(*
TIME		: 2023-11-13 14:59
Version		: 1.0
Creator		: Ulysses
Reference	: IOTA - BLUE
Commecnts	: 按钮功能块，总体和Input差不多，针对按钮做了功能的完善。可以将输入信号强制、反转或延迟
*)
(* 不带延迟 *)
Q			:= ((RawIn OR Force) XOR Invert) AND Enable;
rTrig(CLK:= Q);
Q_RT		:= rTrig.Q;
fTrig(CLK:= Q);
Q_FT		:= fTrig.Q;
Q_Tog	:= NOT (TrigOff AND Enable) AND (Q_RT XOR Q_Tog OR (TrigOn AND Enable));
(* 带延迟 *)
tonDelay(IN:= Q, PT:= DelayTime);
Q_Delay		:= tonDelay.Q;
rTrig_Delay(CLK:= Q_Delay);
Q_Delay_RT	:= rTrig_Delay.Q;
fTrig_Delay(CLK:= Q_Delay);
Q_Delay_FT	:= fTrig_Delay.Q;

Q_Delay_Tog := NOT (TrigOffDelay AND Enable) AND (Q_Delay_RT XOR Q_Delay_Tog OR (TrigOnDelay AND Enable));

END_FUNCTION_BLOCK

// ---- TF11PlcSystem/IO/DI_Input.TcPOU
{attribute 'no_check'}
(* 
按钮功能块 Button
按钮功能块，总体和Input差不多，针对按钮做了功能的完善可以将输入信号强制、反转或延迟
*)
FUNCTION_BLOCK DI_Input
VAR_INPUT
	Invert : BOOL := FALSE; (* False: 不反转Direct \ True: 在源头反转输入Invert Input *)
	ForceOn : BOOL; (* 将输入强制为True, Force the In signal to True *)
	ForceOff : BOOL; (* 将输入强制为True, Force the In signal to True *)
	DelayTime : TIME := T#50MS; (* 延迟输出时间，T#0MS代表无延迟，也可充当滤波功能 *)
	LED AT%Q* : BOOL; (* 如果按钮有LED，绑定到LED的输出上，功能块内部本身不控制LED，需要外部程序通过该输入引脚控制 *)
END_VAR
VAR_OUTPUT
	Q : BOOL;(* 直接输出信号 *)
	QRT : BOOL;(* 输入信号的上升沿 *)
	QFT : BOOL;(* 输入信号的下降沿 *)
	RawIn AT%I* :BOOL; (* 原始输入信号，未经强制、反转及延时 *) 
END_VAR
VAR
	rTrig, rTrig_Delay : R_TRIG;
	fTrig, fTrig_Delay : F_TRIG;
	DelayIn : TON;
	_InternalIn : BOOL;
END_VAR

(*
TIME		: 2024-01-19 17:02
Version		: 1.0
Creator		: Ulysses
Reference	: IOTA - BLUE
Commecnts	: 按钮功能块简化
*)
DelayIn(IN:= RawIn, PT:= DelayTime);
IF DelayTime = T#0S THEN
	(* 不带延迟 *)
	_InternalIn := RawIn;
ELSE
	(* 带延迟 *)
	_InternalIn := DelayIn.Q;
END_IF
Q := ((_InternalIn OR ForceOn) XOR Invert) AND NOT ForceOff;
rTrig(CLK:= Q);
fTrig(CLK:= Q);
QRT := rTrig.Q;
QFT := fTrig.Q;

END_FUNCTION_BLOCK

// ---- TF11PlcSystem/IO/Input.TcPOU
{attribute 'no_check'}
(* 
输入功能块 DI_Input
输入功能块，可以将输入信号强制、反转或延迟，和按钮差不多，默认延迟为0
*)
FUNCTION_BLOCK Input
VAR_INPUT
	Enable : BOOL := TRUE; (* 默认为True, False:不启用,除LED外输入无效  \ True:启用 *)
	Invert : BOOL := FALSE; (* False: 不反转Direct \ True: 在源头反转输入Invert Input *)
	Force : BOOL; (* 将输入强制为True, Force the In signal to True *)
	TrigOnDelay : BOOL; (* 手动将延迟后的Toggle模式输出置为True, 复位优先 *)
	TrigOffDelay : BOOL; (* 手动将延迟后的Toggle模式输出置为False, 复位优先 *)
	DelayTime : TIME := T#0MS; (* 延迟输出时间，默认为T#0MS，代表无延迟 *)

END_VAR
VAR_OUTPUT
	Q_NoDelay : BOOL;(* 直接输出信号 *)
	Q : BOOL;(* 经过延迟后的输出信号,默认延迟0 *)
	Q_RT : BOOL;(* 经过延迟后的输出信号的上升沿,默认延迟0 *)
	Q_FT : BOOL;(* 经过延迟后的输出信号的上升沿,默认延迟0 *)
	Q_Tog : BOOL;(* 经过延迟后的Toggle模式输出,默认延迟0,按一下切换为True，再按一下切换为False *)
	RawIn AT%I* :BOOL; (* 原始输入信号，未经强制、反转及延时 *) 
END_VAR
VAR
	rTrig_Delay : R_TRIG;
	fTrig_Delay : F_TRIG;
	tonDelay : TON;
END_VAR

(*
TIME		: 2023-11-15 17:44
Version		: 1.0
Creator		: Ulysses
Reference	: IOTA - BLUE
Commecnts	: 输入功能块，可以将输入信号强制、反转或延迟，和按钮功能块差不多
*)
(* 不带延迟 *)
Q_NoDelay			:= ((RawIn OR Force) XOR Invert) AND Enable;

(* 带延迟 *)
tonDelay(IN:= Q_NoDelay, PT:= DelayTime);
Q		:= tonDelay.Q;
rTrig_Delay(CLK:= Q);
Q_RT	:= rTrig_Delay.Q;
fTrig_Delay(CLK:= Q);
Q_FT	:= fTrig_Delay.Q;

Q_Tog := NOT (TrigOffDelay AND Enable) AND (Q_RT XOR Q_Tog OR (TrigOnDelay AND Enable));

END_FUNCTION_BLOCK

// ---- TF11PlcSystem/IO/Output.TcPOU
{attribute 'no_check'}
(* 
输出功能块 Output
输出功能块
*)
FUNCTION_BLOCK Output
VAR_INPUT
	Enable : BOOL := TRUE; (* False: 不启用, True: 启用 *)
END_VAR
VAR_OUTPUT
	Out AT%Q* : BOOL; (* 绑定到输出变量，或者利用功能块引脚直接输出 *)
END_VAR
VAR
	InternCycleCounter : UDINT; (* 执行时内置的循环数 *)
	ThisCycleExecuteCounter : UDINT; (* 当前周期循环数 *)
	LastCycleExecuteCounter : UDINT; (* 上个周期循环数 *)
END_VAR

(*
TIME		: 2023-11-13 15:46
Version		: 1.0
Creator		: Ulysses
Reference	: IOTA - BLUE
Commecnts	: 输出功能块，Set返回值代表当前周期调用次数，LastCounter代表上个周期调用次数。
*)

(* 上周期调用次数 *)
PROPERTY LastCounter : UDINT
GET
LastCounter := LastCycleExecuteCounter;
END_GET
END_PROPERTY

(* 返回值代表当前周期内SetOn或者SetOff被执行的次数，正常为1，如果大于1则可能出现双线圈问题 *)
METHOD SetOff : UDINT
VAR_INPUT
END_VAR
VAR
	TempCycleCounter : UDINT;
END_VAR
Out := Enable AND FALSE;
TempCycleCounter := _TaskInfo[GETCURTASKINDEXEX()].CycleCount;
IF InternCycleCounter <> TempCycleCounter THEN
	InternCycleCounter := TempCycleCounter;
	LastCycleExecuteCounter := ThisCycleExecuteCounter;
	ThisCycleExecuteCounter := 0 ;
END_IF
ThisCycleExecuteCounter := ThisCycleExecuteCounter + 1;

SetOff := ThisCycleExecuteCounter;
END_METHOD

(* 返回值代表当前周期内SetOn或者SetOff被执行的次数，正常为1，如果大于1则可能出现双线圈问题 *)
METHOD SetOn : UDINT
VAR_INPUT
END_VAR
VAR
	TempCycleCounter : UDINT;
END_VAR
Out := Enable AND TRUE;
TempCycleCounter := _TaskInfo[GETCURTASKINDEXEX()].CycleCount;
IF InternCycleCounter <> TempCycleCounter THEN
	InternCycleCounter := TempCycleCounter;
	LastCycleExecuteCounter := ThisCycleExecuteCounter;
	ThisCycleExecuteCounter := 0 ;
END_IF
ThisCycleExecuteCounter := ThisCycleExecuteCounter + 1;

SetOn := ThisCycleExecuteCounter;
END_METHOD

END_FUNCTION_BLOCK

// ---- TF11PlcSystem/Logger/ULogger.TcPOU
{attribute 'enable_dynamic_creation'}
FUNCTION_BLOCK ULogger
VAR_INPUT
	bEnable : BOOL;
	bReset : BOOL;
	nBufferSizeSet : UDINT;
	bEnableEventLogger : BOOL;
	bEnableFileLogger : BOOL;
	eSplitLogFileMode : E_LogFileSplitMode := E_LogFileSplitMode.eSplitByDay;
	sLogFilePath : T_MaxString := 'C:\';
	tAutoSave : TIME := T#3M;
END_VAR
VAR_OUTPUT
END_VAR
VAR
	pBufferUsing : POINTER TO BYTE;
	pBufferSaving : POINTER TO BYTE;
	nBufferTotalSize : UDINT;
	nBufferUsedSize : UDINT;
	nBufferSaveSize : UDINT;
	tStartUse : TIME;
	
	bWriteFileRequest : BOOL;
	
	stepWriteFile : INT;
	hFile : UINT;
	fbFileOpen : FB_FileOpen;
	fbFileWrite : FB_FileWrite;
	fbFileClose : FB_FileClose;
	
	
	sFilePathName : T_MaxString;
	
	bError : BOOL;
	
	tonAutoSave : TON;
	tCycleTime : UDINT;
	tPassedTime : UDINT;
	ttimesave: UDINT;
	ttimesavelmt : UDINT;
END_VAR


AutoSave();

CASE stepWriteFile OF
	0:
	IF bWriteFileRequest AND NOT bError THEN
		stepWriteFile := 10;
	ELSIF bError AND bReset THEN
		fbFileOpen(bExecute:= FALSE);
		fbFileWrite(bExecute:= FALSE);
		fbFileClose(bExecute:= FALSE);
		bError := FALSE;
		IF hFile <> 0 THEN
			stepWriteFile := 30;
		END_IF
	END_IF
	10:
	sFilePathName := HandelLogFilePath(SplitLogFileMode:= eSplitLogFileMode, LogFilePath:= sLogFilePath);

	fbFileOpen(sPathName:= sFilePathName, 
		nMode:= FOPEN_MODEAPPEND OR FOPEN_MODETEXT OR FOPEN_MODEPLUS, 
		bExecute:= TRUE);
	IF NOT fbFileOpen.bBusy THEN
		IF NOT fbFileOpen.bError THEN
			hFile := fbFileOpen.hFile;
			stepWriteFile := 20;
		ELSE
			stepWriteFile := 0;
			bError := TRUE;
		END_IF
		fbFileOpen(bExecute:= FALSE);
	END_IF
	20:
	fbFileWrite(
		hFile:= hFile, 
		pWriteBuff:= pBufferSaving, 
		cbWriteLen:= nBufferSaveSize, 
		bExecute:= TRUE);
	IF NOT fbFileWrite.bBusy THEN
		IF NOT fbFileWrite.bError THEN
			stepWriteFile := 30;
		ELSE
			stepWriteFile := 0;
			bError := TRUE;
		END_IF
		fbFileWrite(bExecute:= FALSE);
	END_IF
	30:
	fbFileClose(
		hFile:= hfile, 
		bExecute:= TRUE);
	IF NOT fbFileClose.bBusy THEN
		IF NOT fbFileClose.bError THEN
			hFile := 0;
			stepWriteFile := 0;
			bWriteFileRequest := FALSE;
		ELSE
			hFile := 0;
			bError := TRUE;
			stepWriteFile := 0;
		END_IF
		fbFileClose(bExecute:= FALSE);
	END_IF
END_CASE

METHOD AutoSave : BOOL
VAR_INPUT
END_VAR
IF tCycleTime = 0 THEN
	tCycleTime := _TaskInfo[GETCURTASKINDEXEX()].CycleTime / 10_000;
END_IF
IF nBufferUsedSize > 0 THEN
	tPassedTime := tPassedTime + tCycleTime;
END_IF

ttimesave := TIME_TO_UDINT(tAutoSave);
ttimesavelmt := LIMIT(60_000, ttimesave, 9999_000);
IF tPassedTime >= ttimesavelmt THEN
	SaveBufferNow();
	tPassedTime := 0;
END_IF
END_METHOD

METHOD CreateBuffer : BOOL
VAR_INPUT
END_VAR
VAR
	pTemp : POINTER TO BYTE;
END_VAR
IF nBufferSizeSet = 0 THEN
	RETURN;
END_IF
IF nBufferSizeSet > nBufferTotalSize THEN
	(* 创建使用中缓冲区 *)
	pTemp := __NEW(BYTE, nBufferSizeSet);
	IF pBufferUsing <>0 THEN
		MEMCPY(destAddr:= pTemp, srcAddr:= pBufferUsing, n:= nBufferTotalSize);
		__DELETE(pBufferUsing);
	END_IF
	pBufferUsing := pTemp;
	
	
	(* 创建保存中缓冲区 *)
	pTemp := __NEW(BYTE, nBufferSizeSet);
	IF pBufferSaving <> 0 THEN
		MEMCPY(destAddr:= pTemp, srcAddr:= pBufferSaving, n:= nBufferTotalSize);
		__DELETE(pBufferSaving);
	END_IF
	pBufferSaving := pTemp;
	
	nBufferTotalSize := nBufferSizeSet;
	CreateBuffer := TRUE;
END_IF
END_METHOD

METHOD FB_exit : BOOL
VAR_INPUT
	bInCopyCode : BOOL; // if TRUE, the exit method is called for exiting an instance that is copied afterwards (online change).
END_VAR

VAR
	pBuffer1: INT;
END_VAR
IF NOT bInCopyCode THEN
	IF pBufferUsing <> 0 THEN
		__DELETE(pBufferUsing);
	END_IF
	IF pBufferSaving <> 0 THEN
		__DELETE(pBufferSaving);
	END_IF
	
END_IF
END_METHOD

METHOD HandelLogFilePath : T_MaxString
VAR_INPUT
	SplitLogFileMode : E_LogFileSplitMode;
	LogFilePath : T_MaxString;
END_VAR

VAR
	timestr: DCTIMESTRUCT;
END_VAR
IF SplitLogFileMode = E_LogFileSplitMode.eDontSplit THEN
	HandelLogFilePath := CONCAT(LogFilePath, 'Log.log');
ELSIF eSplitLogFileMode = E_LogFileSplitMode.eSplitByDay THEN
	HandelLogFilePath := CONCAT(LogFilePath, LEFT(STR:= DCTIME64_TO_STRING(F_GetCurDcTaskTime64()), SIZE:= 10));
	HandelLogFilePath := CONCAT(HandelLogFilePath, '.log');
ELSIF eSplitLogFileMode = E_LogFileSplitMode.eSplitByHour THEN
	HandelLogFilePath := CONCAT(LogFilePath, LEFT(STR:= DCTIME64_TO_STRING(F_GetCurDcTaskTime64()), SIZE:= 13));
	HandelLogFilePath := CONCAT(HandelLogFilePath, '.log');
END_IF
END_METHOD

METHOD SaveBufferNow : BOOL
VAR_INPUT
END_VAR
MEMCPY(destAddr:= pBufferSaving, srcAddr:= pBufferUsing, n:= nBufferTotalSize);
nBufferSaveSize := nBufferUsedSize;
nBufferUsedSize := 0;
bWriteFileRequest := TRUE;
END_METHOD

METHOD WriteData : BOOL
VAR_INPUT
	pData : POINTER TO BYTE;
	nSize : UDINT;
END_VAR
IF pData = 0 OR nSize = 0 THEN
	RETURN;
END_IF
IF nBufferSizeSet > nBufferTotalSize THEN
	IF NOT CreateBuffer() THEN
		RETURN;
	END_IF
END_IF
IF nBufferUsedSize = 0 THEN
	tStartUse := TIME();
	IF nSize > nBufferTotalSize THEN
		RETURN;
	END_IF
END_IF
IF nBufferUsedSize + nSize > nBufferTotalSize THEN
	SaveBufferNow();
END_IF

MEMCPY(destAddr:= pBufferUsing + nBufferUsedSize, srcAddr:= pData, n:= nSize);
tPassedTime := 0;
nBufferUsedSize := nBufferUsedSize + nSize;
WriteData := TRUE;
END_METHOD

METHOD WriteLog : BOOL
VAR_INPUT
	LogStr : T_MaxString;
END_VAR
VAR
	Tempstr : STRING;
END_VAR
Tempstr := CONCAT(Tempstr, LEFT(STR:= DCTIME64_TO_STRING(in:= F_GetActualDcTime64()), SIZE:= 27));
Tempstr := CONCAT(Tempstr, ' : ');
Tempstr := CONCAT(Tempstr, LogStr);
Tempstr := CONCAT(Tempstr, '$R');
WriteData(pData:= ADR(Tempstr), nSize:= INT_TO_UDINT(LEN(Tempstr)));
END_METHOD

END_FUNCTION_BLOCK

// ---- TF11PlcSystem/System/File/FB_File.TcPOU
FUNCTION_BLOCK FB_File
VAR_INPUT
END_VAR
VAR_OUTPUT
END_VAR
VAR
	fbFileOpen : FB_FileOpen;
	fbFileClose : FB_FileClose;
	fbFileLoad : FB_FileLoad;
	fileBuffer : ARRAY[0..99] OF BYTE;
END_VAR

fbFileLoad(
	sNetId:= , 
	sPathName:= 'c:\TEMP\LOG.txt', 
	pReadBuff:= ADR(fileBuffer), 
	cbReadLen:= SIZEOF(fileBuffer), 
	bExecute:= , 
	tTimeout:= , 
	bBusy=> , 
	bError=> , 
	nErrId=> , 
	cbRead=> );

END_FUNCTION_BLOCK

// ---- TF11PlcSystem/System/Pendulum4Tc/Constants.TcPOU
FUNCTION_BLOCK Constants
VAR_INPUT

// Number of X in Y.
YEARS_PER_CENTURY : DINT := 100;
YEARS_PER_DECADE : DINT := 10;
MONTHS_PER_YEAR : DINT := 12;
WEEKS_PER_YEAR : DINT := 52;
DAYS_PER_WEEK : DINT := 7;
HOURS_PER_DAY : DINT := 24;
MINUTES_PER_HOUR : DINT := 60;
SECONDS_PER_MINUTE : DINT := 60;
SECONDS_PER_HOUR : DINT := MINUTES_PER_HOUR * SECONDS_PER_MINUTE;
SECONDS_PER_DAY : DINT := HOURS_PER_DAY * SECONDS_PER_HOUR;
US_PER_SECOND : DINT := 1000000;


// Formats
ATOM : STRING := 'YYYY-MM-DDTHH:mm:ssZ';
COOKIE : STRING := 'dddd, DD-MMM-YYYY HH:mm:ss zz';
ISO8601 : STRING := 'YYYY-MM-DDTHH:mm:ssZ';
ISO8601_EXTENDED : STRING := 'YYYY-MM-DDTHH:mm:ss.SSSSSSZ';
RFC822 : STRING := 'ddd, DD MMM YY HH:mm:ss ZZ';
RFC850 : STRING := 'dddd, DD-MMM-YY HH:mm:ss zz';
RFC1036 : STRING := 'ddd, DD MMM YY HH:mm:ss ZZ';
RFC1123 : STRING := 'ddd, DD MMM YYYY HH:mm:ss ZZ';
RFC2822 : STRING := 'ddd, DD MMM YYYY HH:mm:ss ZZ';
RFC3339 : STRING := ISO8601;
RFC3339_EXTENDED : STRING := ISO8601_EXTENDED;
RSS : STRING := 'ddd, DD MMM YYYY HH:mm:ss ZZ';
W3C : STRING := ISO8601;


EPOCH_YEAR : DINT := 1970;

DAYS_PER_N_YEAR : DINT := 365;
DAYS_PER_L_YEAR : DINT := 366;

USECS_PER_SEC : DINT := 1000000;

SECS_PER_MIN : DINT := 60;
SECS_PER_HOUR : DINT := 60 * SECS_PER_MIN;
SECS_PER_DAY : DINT := SECS_PER_HOUR * 24;

// 400-year chunks always have 146097 days (20871 weeks).
SECS_PER_400_YEARS : DINT := 146097 * SECS_PER_DAY;

// The number OF seconds in an aligned 100-year chunk, FOR those that
// do not begin with a leap year and those that do respectively.
SECS_PER_100_YEARS : ARRAY[0..1] OF DINT := [
    (76 * DAYS_PER_N_YEAR + 24 * DAYS_PER_L_YEAR) * SECS_PER_DAY,
    (75 * DAYS_PER_N_YEAR + 25 * DAYS_PER_L_YEAR) * SECS_PER_DAY
];

// The number OF seconds in an aligned 4-year chunk, FOR those that
// do not begin with a leap year and those that do respectively.
SECS_PER_4_YEARS : ARRAY[0..1] OF DINT := [
    (4 * DAYS_PER_N_YEAR + 0 * DAYS_PER_L_YEAR) * SECS_PER_DAY,
    (3 * DAYS_PER_N_YEAR + 1 * DAYS_PER_L_YEAR) * SECS_PER_DAY
];


// The number of seconds in non-leap and leap years respectively.
SECS_PER_YEAR : ARRAY[0..1] OF DINT := [DAYS_PER_N_YEAR * SECS_PER_DAY, DAYS_PER_L_YEAR * SECS_PER_DAY];

DAYS_PER_YEAR : ARRAY[0..1] OF DINT := [DAYS_PER_N_YEAR, DAYS_PER_L_YEAR];

// The month lengths in non-leap and leap years respectively.
DAYS_PER_MONTHS : ARRAY[0..1] OF ARRAY[0..12] OF DINT := [
    [-1, 31, 28, 31, 30, 31, 30, 31, 31, 30, 31, 30, 31],
    [-1, 31, 29, 31, 30, 31, 30, 31, 31, 30, 31, 30, 31]
];

// The day offsets of the beginning of each (1-based) month in non-leap
// and leap years respectively.
// For example, in a leap year there are 335 days before December.
MONTHS_OFFSETS : ARRAY[0..1] OF ARRAY[0..12] OF DINT := [
    [-1, 0, 31, 59, 90, 120, 151, 181, 212, 243, 273, 304, 334, 365],
    [-1, 0, 31, 60, 91, 121, 152, 182, 213, 244, 274, 305, 335, 366]
];

DAY_OF_WEEK_TABLE : ARRAY[0..11] OF DINT := [0, 3, 2, 5, 0, 3, 5, 1, 4, 6, 2, 4];


TM_SUNDAY : DINT := 0;
TM_MONDAY : DINT := 1;
TM_TUESDAY : DINT := 2;
TM_WEDNESDAY : DINT := 3;
TM_THURSDAY : DINT := 4;
TM_FRIDAY : DINT := 5;
TM_SATURDAY : DINT := 6;

TM_JANUARY : DINT := 0;
TM_FEBRUARY : DINT := 1;
TM_MARCH : DINT := 2;
TM_APRIL : DINT := 3;
TM_MAY : DINT := 4;
TM_JUNE : DINT := 5;
TM_JULY : DINT := 6;
TM_AUGUST : DINT := 7;
TM_SEPTEMBER : DINT := 8;
TM_OCTOBER : DINT := 9;
TM_NOVEMBER : DINT := 10;
TM_DECEMBER : DINT := 11;

END_VAR

END_FUNCTION_BLOCK

// ---- TF11PlcSystem/System/Pendulum4Tc/Functions/F_TzInfoBiasToTzStr.TcPOU
FUNCTION F_TzInfoBiasToTzStr : STRING
VAR_INPUT
	tzBias : DINT;
END_VAR
VAR
	UtcOffset : DINT;
END_VAR

UtcOffset := (0-tzBias) / 60;
IF UtcOffset > 0 AND UtcOffset < 10 THEN
	F_TzInfoBiasToTzStr := CONCAT(STR1:= 'UTC+0', STR2:= DINT_TO_STRING(UtcOffset));
ELSIF UtcOffset >= 10 AND UtcOffset <= 12 THEN
	F_TzInfoBiasToTzStr := CONCAT(STR1:= 'UTC+', STR2:= DINT_TO_STRING(UtcOffset));
ELSIF UtcOffset < 0 AND UtcOffset > -10 THEN
	F_TzInfoBiasToTzStr := CONCAT(STR1:= 'UTC-0', STR2:= DINT_TO_STRING(UtcOffset));
ELSIF UtcOffset <=10 AND UtcOffset >= -12 THEN
	F_TzInfoBiasToTzStr := CONCAT(STR1:= 'UTC-', STR2:= DINT_TO_STRING(UtcOffset));
ELSIF UtcOffset = 0 THEN
	F_TzInfoBiasToTzStr := 'UTC';
END_IF

END_FUNCTION

// ---- TF11PlcSystem/System/Pendulum4Tc/Helper/calcDayNumber.TcPOU
(* 计算某个日期 *)
FUNCTION calcDayNumber : dint
VAR_INPUT
	Year : DINT;
	Month : DINT;
	Day : DINT;
END_VAR
VAR
END_VAR

month := (month + 9) MOD 12;
year := year - month / 10;
calcDayNumber := (
        365 * year
        + year / 4
        - year / 100
        + year / 400
        + (month * 306 + 5) / 10
        + (day - 1)
    );

END_FUNCTION

// ---- TF11PlcSystem/System/Pendulum4Tc/Helper/calcPreciseDiff.TcPOU
FUNCTION calcPreciseDiff : PtPreciseDiff
VAR_INPUT
	D1 : PtDateTime;
	D2 : PtDateTime;
END_VAR
VAR
	HourDiff : DINT;
	
END_VAR

IF isDateTimeEqual(D1, D2) THEN
	calcPreciseDiff.Set(0,0,0,0,0,0,0,0);
	RETURN;
END_IF
calcPreciseDiff.total_days := ABS(calcDayNumber(D1.Year, d1.Month, d1.Day) - calcDayNumber(D2.Year, d2.Month, d2.Day));

END_FUNCTION

// ---- TF11PlcSystem/System/Pendulum4Tc/Helper/PtPreciseDiff.TcPOU
FUNCTION_BLOCK PtPreciseDiff
VAR_INPUT
	years: DINT;
    months: DINT;
    days: DINT;
    hours: DINT;
    minutes: DINT;
    seconds: DINT;
    microseconds: DINT;
    total_days: DINT;
END_VAR
VAR_OUTPUT
END_VAR
VAR
END_VAR

METHOD Set : BOOL
VAR_INPUT
	years: DINT;
    months: DINT;
    days: DINT;
    hours: DINT;
    minutes: DINT;
    seconds: DINT;
    microseconds: DINT;
    total_days: DINT;
END_VAR
THIS^.years := years;
THIS^.months := months;
THIS^.days := days;
THIS^.hours := hours;
THIS^.minutes := minutes;
THIS^.seconds := seconds;
THIS^.microseconds := microseconds;
THIS^.total_days := total_days;
END_METHOD

END_FUNCTION_BLOCK

// ---- TF11PlcSystem/System/Pendulum4Tc/Helper/isDateTimeEqual.TcPOU
FUNCTION isDateTimeEqual : bool
VAR_INPUT
	D1 : PtDateTime;
	D2 : PtDateTime;
END_VAR
VAR
END_VAR

isDateTimeEqual 
:= D1.Year = D2.Year
AND D1.Month = D2.Month
AND D1.Day = D2.Day
AND D1.Hour = D2.Hour
AND D1.Minute = D2.Minute
AND D1.Second = D2.Second
AND D1.Microsecond = D2.Microsecond
AND D1.TimeZone = D2.TimeZone;

END_FUNCTION

// ---- TF11PlcSystem/System/Pendulum4Tc/Helper/isLeapYear.TcPOU
FUNCTION isLeapYear : BOOL
VAR_INPUT
	Year : DINT;
END_VAR
VAR
END_VAR

isLeapYear := (year mod 4 = 0) and ((year mod 100 <> 0) or (year mod 400 = 0));

END_FUNCTION

// ---- TF11PlcSystem/System/Pendulum4Tc/PtHelper.TcPOU
FUNCTION_BLOCK PtHelper
VAR_INPUT
END_VAR
VAR_OUTPUT
END_VAR
VAR
END_VAR

END_FUNCTION_BLOCK

// ---- TF11PlcSystem/System/Pendulum4Tc/PtTimeSource.TcPOU
FUNCTION_BLOCK PtTimeSource IMPLEMENTS I_PtTimesource
VAR_INPUT
END_VAR
VAR_OUTPUT
END_VAR
VAR
	_DateTime : ptDateTime;
	DefaultTimeZoneTime : TIMESTRUCT;
	
END_VAR

METHOD getDateTime : PtDateTime
VAR_INPUT
END_VAR

DefaultTimeZoneTime := FILETIME64_TO_SYSTEMTIME(fileTime:= F_GetSystemTime());
_DateTime.Set(
	Year:= DefaultTimeZoneTime.wYear, 
	Month:= DefaultTimeZoneTime.wMonth, 
	Day:= DefaultTimeZoneTime.wDay, 
	Hour:= DefaultTimeZoneTime.wHour, 
	Minute:= DefaultTimeZoneTime.wMinute, 
	Second:= DefaultTimeZoneTime.wSecond, 
	Microsecond:= DefaultTimeZoneTime.wMilliseconds, 
	TimeZone:= 0);
getDateTime := _DateTime;
END_METHOD

END_FUNCTION_BLOCK

// ---- TF11PlcSystem/System/SystemInfo/System_AppInfo.TcPOU
FUNCTION_BLOCK System_AppInfo
VAR_INPUT
	
END_VAR
VAR_OUTPUT
	ObjectID: UDINT;
	TaskCount: UDINT;
	OnlineChangeCount: UDINT;
	Flags: DWORD;
	AdsPort: UINT;
	BootDataLoaded: BOOL;
	OldBootData: BOOL;
	AppTimestamp: DATE_AND_TIME;
	KeepOutputsOnBreakpoint: BOOL;
	ShutdownInProgress: BOOL;
	LicensePending: BOOL;
	BlueScreenOccured: BOOL;
	LoggedIn: BOOL;
	PersistentStatus: EPlcPersistentStatus;
	TcComSrvPointer: ITComObjectServer;
	AppName: STRING(63);
	ProjectName: STRING(63);
END_VAR
VAR
	(* AppInfo Source Data *)
	_ThisAppInfo: PlcAppSystemInfo;
	
END_VAR

_ThisAppInfo := TwinCAT_SystemInfoVarList._AppInfo;
ObjectID := _ThisAppInfo.ObjId;
TaskCount := _ThisAppInfo.TaskCnt;
OnlineChangeCount := _ThisAppInfo.OnlineChangeCnt;
Flags := _ThisAppInfo.Flags;
AdsPort := _ThisAppInfo.AdsPort;
BootDataLoaded := _ThisAppInfo.BootDataLoaded;
OldBootData := _ThisAppInfo.OldBootData;
AppTimestamp := _ThisAppInfo.AppTimestamp;
KeepOutputsOnBreakpoint := _ThisAppInfo.KeepOutputsOnBP;
ShutdownInProgress := _ThisAppInfo.ShutdownInProgress;
LicensePending := _ThisAppInfo.LicensesPending;
BlueScreenOccured := _ThisAppInfo.BSODOccured;
LoggedIn := _ThisAppInfo.LoggedIn;
PersistentStatus := _ThisAppInfo.PersistentStatus;
TcComSrvPointer := _ThisAppInfo.TComSrvPtr;
AppName := _ThisAppInfo.AppName;
ProjectName := _ThisAppInfo.ProjectName;

END_FUNCTION_BLOCK

// ---- TF11PlcSystem/System/SystemInfo/System_IpcInfo.TcPOU
FUNCTION_BLOCK System_IpcInfo
VAR_INPUT
END_VAR
VAR_OUTPUT
END_VAR
VAR
END_VAR

END_FUNCTION_BLOCK

// ---- TF11PlcSystem/System/SystemInfo/System_TaskInfo.TcPOU
FUNCTION_BLOCK System_TaskInfo
VAR_INPUT
	
END_VAR
VAR_OUTPUT
	// Object ID of the task reference, from which the PLC program is called.
	ObjId: UDINT;
	// Set task cycle time in multiples of 100 ns
	CycleTime: UDINT;
	// Set task priority
	Priority: UINT;
	// ADS port of the task
	AdsPort: UINT;
	(* 
	Cycle counter
	Please note that the cycle counter refers to the actual system task 
	and not to the task reference of the PLC project. The background to 
	this is that several PLC projects or other TcCOM modules can share 
	a task and these modules can thus access the same cycle counter. 
	As a result, the cycle counter is reset during a TwinCAT restart in 
	RUN mode (and not when resetting the PLC project). *)
	CycleCount: UDINT;
	// Distributed Clock System Time. It remains constant for a task runtime.
	DcTaskTime: LINT;
	// Cycle time required for the last cycle in multiples of 100 ns
	LastExecTime: UDINT;
	// During the first PLC task cycle, this variable has the value TRUE.
	FirstCycle: BOOL;
	(* 
	This variable indicates whether the set task cycle time was exceeded.
	The value of the CycleTimeExceeded variable is updated in each cycle. 
	The variable is set to 0 if the previous cycle has been completed 
	within its intended timeframe, otherwise to 1. *)
	CycleTimeExceeded: BOOL;
	(* 
	This variable has the value TRUE if the origin of the current call 
	is declared with the attribute 'TcCallAfterOutputUpdate'. *)
	InCallAfterOutputUpdate: BOOL;
	(* This variable has the value TRUE if the real-time limit is 
	exceeded on a mixed core (Windows + real-time on one core). In this 
	case the value TRUE refers to the core on which the corresponding 
	task is running. *)
	RTViolation: BOOL;
	// Name of the task reference object in the PLC project (e.g. 'MyPlcProject_PlcTaskRef')
	TaskName: STRING(63);
END_VAR
VAR
	
	_ThisTaskInfo: PlcTaskSystemInfo;
	_AllTaskInfo : ARRAY[0..10] OF PlcTaskSystemInfo;
	index : UDINT;
	TaskCount : UDINT;
	TaskIndex : DINT ;
	
	
END_VAR

TaskCount := _AppInfo.TaskCnt;
FOR index := 1 TO LIMIT(1,TaskCount,10)  DO
	_AllTaskInfo[index] := _TaskInfo[index];
END_FOR
TaskIndex := GETCURTASKINDEXEX();
_ThisTaskInfo := _AllTaskInfo[TaskIndex];

_ThisTaskInfo := _TaskInfo[TaskIndex];
ObjId := _ThisTaskInfo.ObjId; 
CycleTime := _ThisTaskInfo.CycleTime;
Priority := _ThisTaskInfo.Priority;
AdsPort := _ThisTaskInfo.AdsPort;
CycleCount := _ThisTaskInfo.CycleCount;
DcTaskTime := _ThisTaskInfo.DcTaskTime;
LastExecTime := _ThisTaskInfo.LastExecTime;
FirstCycle := _ThisTaskInfo.FirstCycle;
CycleTimeExceeded := _ThisTaskInfo.CycleTimeExceeded;
InCallAfterOutputUpdate := _ThisTaskInfo.InCallAfterOutputUpdate;
RTViolation := _ThisTaskInfo.RTViolation;

TaskName := _ThisTaskInfo.TaskName;

METHOD getCurrentTaskInfo : REFERENCE TO PlcTaskSystemInfo
VAR_INPUT
END_VAR
getCurrentTaskInfo REF= _ThisTaskInfo;
END_METHOD

METHOD getTaskCount : UDINT
VAR_INPUT
END_VAR
getTaskCount := _AppInfo.TaskCnt;
END_METHOD

METHOD getTaskFirstIndex : UDINT
VAR_INPUT
END_VAR
getTaskFirstIndex := 1;
END_METHOD

METHOD getTaskInfoByIndex : REFERENCE TO PlcTaskSystemInfo
VAR_INPUT
	Index : UDINT;
END_VAR
IF Index >= 1 AND index <= 10 THEN
	getTaskInfoByIndex REF= _AllTaskInfo[Index];
ELSE
	getTaskInfoByIndex REF= _AllTaskInfo[0];
END_IF
END_METHOD

END_FUNCTION_BLOCK

// ---- TF11PlcSystem/System/SystemPulses.TcPOU
{attribute 'no_check'}
(* 
系统脉冲 System Pulse
提供了一些基础的脉冲，包含西门子M0.0-M0.7的脉冲，通过Property调用
*)
FUNCTION_BLOCK SystemPulses
VAR_INPUT
	EnableAll : BOOL := TRUE;
END_VAR
VAR_OUTPUT
END_VAR
VAR
	_T40ms : Pulse := (bEnable:= TRUE, Time_On:=T#20MS, Time_Off:=T#20MS);
	_T100ms : Pulse := (bEnable:= TRUE, Time_On:=T#50MS, Time_Off:=T#50MS);(* 周期:100ms, 频率:10Hz, M0.0 *)
	_T200ms : Pulse := (bEnable:= TRUE, Time_On:=T#100MS, Time_Off:=T#100MS);(* 周期:200ms, 频率:5Hz, M0.1 *)
	_T400ms : Pulse := (bEnable:= TRUE, Time_On:=T#200MS, Time_Off:=T#200MS);(* 周期:400ms, 频率:2.5Hz, M0.2 *)
	_T500ms : Pulse := (bEnable:= TRUE, Time_On:=T#250MS, Time_Off:=T#250MS);(* 周期:500ms, 频率:2Hz, M0.3 *)
	_T800ms : Pulse := (bEnable:= TRUE, Time_On:=T#400MS, Time_Off:=T#400MS);(* 周期:800ms, 频率:1.25Hz, M0.4 *)
	_T1s : Pulse := (bEnable:= TRUE, Time_On:=T#500MS, Time_Off:=T#500MS);(* 周期:1s, 频率:1Hz, M0.5 *)
	_T1s600ms : Pulse := (bEnable:= TRUE, Time_On:=T#800MS, Time_Off:=T#800MS);(* 周期:1.6s, 频率:0.625Hz, M0.6 *)
	_T2s : Pulse := (bEnable:= TRUE, Time_On:=T#1S, Time_Off:=T#1S);(* 周期:2s, 频率:0.5Hz, M0.7 *)
	_T5s : Pulse := (bEnable:= TRUE, Time_On:=T#2500MS, Time_Off:=T#2500MS);(* 周期:5s, 频率:0.2Hz *)
	_T10s : Pulse := (bEnable:= TRUE, Time_On:=T#5S, Time_Off:=T#5S);(* 周期:10s, 频率:0.1Hz *)
	_T30s : Pulse := (bEnable:= TRUE, Time_On:=T#15S, Time_Off:=T#15S);(* 周期:30s, 频率: *)
	_T1m : Pulse := (bEnable:= TRUE, Time_On:=T#30S, Time_Off:=T#30S);(* 周期:1m, 频率: *)
	_T5m : Pulse := (bEnable:= TRUE, Time_On:=T#150S, Time_Off:=T#150S);(* 周期:5m, 频率: *)
	_T10m : Pulse := (bEnable:= TRUE, Time_On:=T#300S, Time_Off:=T#300S);(* 周期:10m, 频率: *)
	_T60m : Pulse := (bEnable:= TRUE, Time_On:=T#30M, Time_Off:=T#30M);(* 周期:60m, 频率: *)
END_VAR

(* 
Title		: 系统脉冲 System Pulse
Time		: 2023-11-13 13:25
Version		: 1.0
Creator		: Ulysses
Reference	: IOTA - Blue \ Siemens
Commecnts	: 提供了一些基础的脉冲，包含西门子M0.0-M0.7的脉冲
*)
IF EnableAll THEN
	_T40ms(Q=> , RT=> , FT=> );
	_T100ms(Q=> , RT=> , FT=> );
	_T200ms(Q=> , RT=> , FT=> );
	_T400ms(Q=> , RT=> , FT=> );
	_T500ms(Q=> , RT=> , FT=> );
	_T800ms(Q=> , RT=> , FT=> );
	_T1s(Q=> , RT=> , FT=> );
	_T1s600ms(Q=> , RT=> , FT=> );
	_T2s(Q=> , RT=> , FT=> );
	_T5s(Q=> , RT=> , FT=> );
	_T10s(Q=> , RT=> , FT=> );
	_T30s(Q=> , RT=> , FT=> );
	_T1m(Q=> , RT=> , FT=> );
	_T5m(Q=> , RT=> , FT=> );
	_T10m(Q=> , RT=> , FT=> );
	_T60m(Q=> , RT=> , FT=> );
END_IF

PROPERTY T100ms : bool
GET
T100ms := _T100ms.Q;
END_GET
END_PROPERTY

PROPERTY T10m : BOOL
GET
T10m := _T10m.Q;
END_GET
END_PROPERTY

PROPERTY T10s : BOOL
GET
T10s := _T10s.Q;
END_GET
END_PROPERTY

PROPERTY T1m : BOOL
GET
T1m := _T1m.Q;
END_GET
END_PROPERTY

PROPERTY T1s : BOOL
GET
T1s := _T1s.Q;
END_GET
END_PROPERTY

PROPERTY T1s600ms : BOOL
GET
T1s600ms := _T1s600ms.Q;
END_GET
END_PROPERTY

PROPERTY T200ms : BOOL
GET
T200ms := _T200ms.Q;
END_GET
END_PROPERTY

PROPERTY T2s : BOOL
GET
T2s := _T2s.Q;
END_GET
END_PROPERTY

PROPERTY T30s : BOOL
GET
T30s := _T30s.Q;
END_GET
END_PROPERTY

PROPERTY T400ms : BOOL
GET
T400ms := _T400ms.Q;
END_GET
END_PROPERTY

PROPERTY T40ms : bool
GET
T40ms := _T40ms.Q;
END_GET
END_PROPERTY

PROPERTY T500ms : BOOL
GET
T500ms := _T500ms.Q;
END_GET
END_PROPERTY

PROPERTY T5m : BOOL
GET
T5m := _T5m.Q;
END_GET
END_PROPERTY

PROPERTY T5s : BOOL
GET
T5s := _T5s.Q;
END_GET
END_PROPERTY

PROPERTY T60m : BOOL
GET
T60m := _T60m.Q;
END_GET
END_PROPERTY

PROPERTY T800ms : BOOL
GET
T800ms := _T800ms.Q;
END_GET
END_PROPERTY

END_FUNCTION_BLOCK

// ---- TF11PlcSystem/System/Time/FunctionBlocks/Pulse.TcPOU
{attribute 'no_check'}
(* 
脉冲生成器 Pulse Generator
设定On\Off时间，生成指定的脉冲
*)
FUNCTION_BLOCK Pulse
VAR_INPUT
	bEnable					: BOOL	:= FALSE;	(*开始*)
	Time_On : TIME; (* TIME, On脉冲时间, 最小时间为扫描周期两倍 *)
	Time_Off : TIME; (* TIME, Off脉冲时间, 最小时间为扫描周期两倍 *)
END_VAR
VAR_OUTPUT
	Q	: BOOL; (* BOOL, 脉冲输出 *)
	RT	: BOOL; (* BOOL, 脉冲输出上升沿 *)
	FT	: BOOL; (* BOOL, 脉冲输出下降沿 *)
END_VAR
VAR
	TonOff, TonOn				: TON;
	rTrig	: R_TRIG;
	fTrig	: F_TRIG;
	
END_VAR

(* 
Title		: 脉冲生成器 Pulse Generator
Time		: 2023-11-13 13:26
Version		: 1.0
Creator		: Ulysses
Reference	: Beckhoff_GZ - Lib_Basic
Commecnts	: 这个程序生成的脉冲就不会受到扫描周期的影响, On\Off信号最小时间为扫描周期两倍，即最小脉冲周期为扫描周期四倍
*)
;
(* tonOn出发 *)
TonOff(IN := bEnable, PT := Time_Off);
TonOn(IN := TonOff.Q, PT := Time_On);
IF TonOn.Q THEN
(* 当计时器2输出信号时，复位并重启计时器1 *)
	TonOff(IN := FALSE);
	TonOff(IN := bEnable, PT := Time_On);
END_IF
(* 输出必须放在最后，不然会导致On信号多一个周期，Off信号少一个周期 *)
Q := TonOff.Q;
rTrig(CLK:= TonOff.Q, Q=> RT);
fTrig(CLK:= TonOff.Q, Q=> FT);

END_FUNCTION_BLOCK

// ---- TF11PlcSystem/System/Time/FunctionBlocks/FB_TimeConvertorM.TcPOU
{attribute 'hide_all_locals'}
{attribute 'no_check'}
(* 
时间转换 FB_TimeConvertorM
用于在多种常用的时间格式间进行转换的功能块,不考虑时区
*)
FUNCTION_BLOCK FB_TimeConvertorM
VAR_INPUT
	InputType : UDINT := 0 ; (* 0:DcTaskTime 1:10位Unix 2:13位Unix 3:FileTime64 4:DateAndTime 5:SystemTime *)
	iDcTaskTime : LINT; (* DcTaskTime从2000-01-01 00:00:00:000开始，精确到1ns *)
	iUnixTimeStamp10 : ULINT; (* 10位unix时间戳，代表从格林威治时间1970-01-01 00:00:00开始的秒数 *)
	iUnixTimeStamp13 : ULINT; (* 13位unix时间戳，代表从格林威治时间1970-01-01 00:00:00开始的秒数+3位毫秒数 *)
	iFileTime64 : T_FILETIME64; (* Utilities库中引入的Windows文件系统时间戳，代表从格林威治时间1601-01-01 00:00:00开始的纳秒数 *)
	iDateAndTime : DATE_AND_TIME; (* TwinCAT系统自带的本地时间日期格式，数值为10位unix时间戳，受到时区影响 *)
	iSystemTime : TIMESTRUCT; (* Utilities库中定义的本地时间日期格式，包含了年月日时分秒毫秒的结构体，受到时区影响 *)
END_VAR
VAR_OUTPUT
	oDcTaskTime : LINT;(* DcTaskTime从2000-01-01 00:00:00:000开始，精确到1ns *)
	oUnixTimeStamp10 : ULINT; (* 10位unix时间戳，代表从格林威治时间1970-01-01 00:00:00开始的秒数 *)
	oUnixTimeStamp13 : ULINT; (* 13位unix时间戳，代表从格林威治时间1970-01-01 00:00:00开始的秒数+3位毫秒数 *)
	oFileTime64 : T_FILETIME64; (* Utilities库中引入的Windows文件系统时间戳，代表从格林威治时间1601-01-01 00:00:00开始的纳秒数 *)
	oDateAndTime : DATE_AND_TIME; (* TwinCAT系统自带的本地时间日期格式，数值为10位unix时间戳，受到时区影响 *)
	oSystemTime : TIMESTRUCT; (* Utilities库中定义的本地时间日期格式，包含了年月日时分秒毫秒的结构体，受到时区影响 *)
	oStringTime : STRING(23); (* 时间字符串，年月日时分秒毫秒 *)
	oStringDate : STRING(10); (* 时间字符串，年月日 *)
	oStringTimeOfDay : STRING(12); (* 时间字符串，时分秒毫秒 *)
END_VAR
VAR
END_VAR

(* 测试数据751214127491000000,1697898927,1697898927491,LDT#2023-10-21-14:35:22.491,DT#2023-10-21-14:35:22,..  *)
(* 由于Utilities库中自带了Filetime64与DT, Systemtime之间的转换，本功能块仅仅是添加了Filetime64与DcTaskTime与UnixTimeStamp之前的转换 *)
(* 转换思路是先尽可能转换成Filetime64，再利用自带函数转换 *)
(* Filetime64与DcTaskTime与UnixTimeStamp都是一种时间戳，区别在于起始时间或精度各不相同 *)
(* DcTaskTime从2000-01-01 00:00:00:000开始，精确到1ns *)
(* 10位Unix时间戳从1970-01-01 00:00:00开始，精确到1s，13位Unix时间戳加了三位表示毫秒的数 *)
(* FileTime64从1601-01-01 00:00:00开始，精确到100ns, *)
(* 946684800:从1970-2000年的秒数  11644473600:从1601-1970的秒数  5:误差补偿 *)
CASE InputType OF
	0:(* DcTaskTime从2000-01-01 00:00:00:000开始，精确到1ns *)
	(* Input *)
	oDcTaskTime := iDcTaskTime;
	(* Convert *)
	oFileTime64 := LINT_TO_ULINT(oDcTaskTime)/100 + 946684800_0000000 + 11644473600_0000000 (*- 5_0000000*);
	oUnixTimeStamp13 := oFileTime64/10000 (*+ 5000 *)- 11644473600000;
	oUnixTimeStamp10 := oUnixTimeStamp13 / 1000;
	oDateAndTime := FILETIME64_TO_DT(oFileTime64);
	oSystemTime := FILETIME64_TO_SYSTEMTIME(oFileTime64);
	
	1: (* Unix10 -> Unix13 : 由于10位时间戳不包含毫秒，所以转换出来的也不包含 *)
	(* Input *)
	oUnixTimeStamp10 := iUnixTimeStamp10;
	(* Convert *)
	oUnixTimeStamp13 := oUnixTimeStamp10 * 1000;
	oFileTime64 := (oUnixTimeStamp13 + 11644473600000 (*- 5000*)) * 10000;
	oDateAndTime := FILETIME64_TO_DT(oFileTime64);
	oSystemTime := FILETIME64_TO_SYSTEMTIME(oFileTime64);
	oDcTaskTime := ULINT_TO_LINT(oFileTime64 - 946684800_0000000 - 11644473600_0000000 (*+ 5_0000000*)) * 100;
	
	2:
	(* Input *)
	oUnixTimeStamp13 := iUnixTimeStamp13;
	(* Convert *)
	oUnixTimeStamp10 := oUnixTimeStamp13 / 1000;
	oFileTime64 := (oUnixTimeStamp13 + 11644473600000 (*- 5000*)) * 10000;
	oDateAndTime := FILETIME64_TO_DT(oFileTime64);
	oSystemTime := FILETIME64_TO_SYSTEMTIME(oFileTime64);
	oDcTaskTime := ULINT_TO_LINT(oFileTime64 - 946684800_0000000 - 11644473600_0000000 (*+ 5_0000000*)) * 100;
	
	3:
	(* Input *)
	oFileTime64 := iFileTime64;
	(* Convert *)
	oUnixTimeStamp13 := oFileTime64/10000 (*+ 5000*) - 11644473600000;
	oUnixTimeStamp10 := oUnixTimeStamp13 / 1000;
	oDateAndTime := FILETIME64_TO_DT(oFileTime64);
	oSystemTime := FILETIME64_TO_SYSTEMTIME(oFileTime64);
	oDcTaskTime := ULINT_TO_LINT(oFileTime64 - 946684800_0000000 - 11644473600_0000000 (*+ 5_0000000*)) * 100;
	
	4:
	(* Input *)
	oDateAndTime := iDateAndTime;
	(* Convert *)
	oFileTime64 := DT_TO_FILETIME64(oDateAndTime);
	oUnixTimeStamp13 := oFileTime64/10000 (*+ 5000*) - 11644473600000;
	oUnixTimeStamp10 := oUnixTimeStamp13 / 1000;
	oSystemTime := FILETIME64_TO_SYSTEMTIME(oFileTime64);
	oDcTaskTime := ULINT_TO_LINT(oFileTime64 - 946684800_0000000 - 11644473600_0000000 (*+ 5_0000000*)) * 100;
	
	5:
	(* Input *)
	oSystemTime :=iSystemTime;
	(* Convert *)
	oFileTime64 := SYSTEMTIME_TO_FILETIME64(oSystemTime);
	oUnixTimeStamp13 := oFileTime64/10000 (*+ 5000*) - 11644473600000;
	oUnixTimeStamp10 := oUnixTimeStamp13 / 1000;
	oDateAndTime := FILETIME64_TO_DT(oFileTime64);
	oDcTaskTime := ULINT_TO_LINT(oFileTime64 - 946684800_0000000 - 11644473600_0000000 (*+ 5_0000000*)) * 100;
	
END_CASE
(* 2023-10-21 15:18:31:771 *)
oStringTime := F_SYSTEMTIME_TO_String6(oSystemTime, '');
oStringDate := MID(STR:= oStringTime, LEN:= 10, POS:= 1);
oStringTimeOfDay := MID(STR:= oStringTime, LEN:= 12, POS:= 12);

END_FUNCTION_BLOCK

// ---- TF11PlcSystem/System/Time/Functions/F_SYSTEMTIME_TO_String6.TcPOU
FUNCTION F_SYSTEMTIME_TO_String6 : String
VAR_INPUT
	SYSTEMTIME : TIMESTRUCT;
	TimeFormat : STRING := '%s-%s-%s %s:%s:%s:%s';
END_VAR
VAR
	fbFormatString : FB_FormatString;
END_VAR

IF TimeFormat = '' THEN
	TimeFormat := '%.4d-%.2d-%.2d %.2d:%.2d:%.2d:%.3d';
END_IF
fbFormatString(
	sFormat:= TimeFormat, 
	arg1:= F_WORD(SYSTEMTIME.wYear), 
	arg2:= F_WORD(SYSTEMTIME.wMonth), 
	arg3:= F_WORD(SYSTEMTIME.wDay), 
	arg4:= F_WORD(SYSTEMTIME.wHour), 
	arg5:= F_WORD(SYSTEMTIME.wMinute), 
	arg6:= F_WORD(SYSTEMTIME.wSecond), 
	arg7:= F_WORD(SYSTEMTIME.wMilliseconds), 
	arg8:= , 
	arg9:= , 
	arg10:= , 
	bError=> , 
	nErrId=> , 
	sOut=> F_SYSTEMTIME_TO_String6);

END_FUNCTION

// ---- TF11PlcSystem/System/Time/FunctionBlocks/FB_Time_Task.TcPOU
FUNCTION_BLOCK FB_Time_Task
VAR_INPUT
END_VAR
VAR_OUTPUT
	(* AppInfo *)
	oTaskInfo: PlcTaskSystemInfo;
	oAppInfo: PlcAppSystemInfo;
	(* Time *)
	oDcTaskTime: LINT;
	oUnixTimeStamp10: ULINT;
	oUnixTimeStamp13: ULINT;
	oFileTime64: ULINT;
	oDateAndTime: DATE_AND_TIME;
	oSystemTime: TIMESTRUCT;
	oStringTime: STRING;
	oStringDate: STRING;
	oStringTimeOfDay: STRING;
END_VAR
VAR
	fbTimeConvertor : FB_TimeConvertorM;
END_VAR

(* 
Title		: 系统时间 FB_Time_Task
Time		: 2023-11-13 13:25
Version		: 1.0
Creator		: Ulysses
Reference	: IOTA - Blue \ Siemens
Commecnts	: 从Task数据获取DcTaskTime，并通过转换功能块转换为其他格式
*)
oAppInfo := _AppInfo;
oTaskInfo := _TaskInfo[GETCURTASKINDEXEX()];
fbTimeConvertor(
	InputType:= 0, 
	iDcTaskTime:= _TaskInfo[GETCURTASKINDEXEX()].DcTaskTime, 
	oDcTaskTime=> oDcTaskTime, 
	oUnixTimeStamp10=> oUnixTimeStamp10, 
	oUnixTimeStamp13=> oUnixTimeStamp13, 
	oFileTime64=> oFileTime64, 
	oDateAndTime=> oDateAndTime, 
	oSystemTime=> oSystemTime, 
	oStringTime=> oStringTime, 
	oStringDate=> oStringDate, 
	oStringTimeOfDay=> oStringTimeOfDay);

END_FUNCTION_BLOCK

// ---- TF11PlcSystem/System/Time/FunctionBlocks/TimeConvertor.TcPOU
FUNCTION_BLOCK TimeConvertor
VAR_INPUT
END_VAR
VAR_OUTPUT
END_VAR
VAR
END_VAR

METHOD fromfiletime64 : ST_TimeConvertor
VAR_INPUT
END_VAR
END_METHOD

END_FUNCTION_BLOCK

// ---- TF11PlcSystem/System/Time/Functions/F_FormatTime.TcPOU
FUNCTION F_FormatTime : STRING
VAR_INPUT
	TimeFormat : STRING;
	TimeInput : TIMESTRUCT;
END_VAR
VAR
	POS_YYYY : INT;
	POS_MM : INT;
	POS_DD : INT;
	POS_hh : INT;
	POS_Lmm : INT;
	POS_ss : INT;
	POS_xxx : INT;
	YYYY : STRING(4);
	MM : STRING(2);
	DD : STRING(2);
	hh : STRING(2);
	Lmm : STRING(2);
	ss : STRING(2);
	xxx : STRING(3);
	TEMPSTRING : STRING;
END_VAR

POS_YYYY := FIND(STR1:= TimeFormat, STR2:= 'YYYY');
POS_MM := FIND(STR1:= TimeFormat, STR2:= 'MM');
POS_DD := FIND(STR1:= TimeFormat, STR2:= 'DD');
POS_hh := FIND(STR1:= TimeFormat, STR2:= 'hh');
POS_Lmm := FIND(STR1:= TimeFormat, STR2:= 'mm');
POS_ss := FIND(STR1:= TimeFormat, STR2:= 'ss');
POS_xxx := FIND(STR1:= TimeFormat, STR2:= 'xxx');

YYYY := TO_STRING(TimeInput.wYear);
MM := TO_STRING(TimeInput.wMonth);
DD := TO_STRING(TimeInput.wDay);
hh := TO_STRING(TimeInput.wHour);
Lmm := TO_STRING(TimeInput.wMinute);
ss := TO_STRING(TimeInput.wSecond);
xxx := TO_STRING(TimeInput.wMilliseconds);
WHILE LEN(YYYY) < 4 DO
	YYYY := CONCAT(STR1:= '0', STR2:= YYYY);
END_WHILE;
WHILE LEN(MM) < 2 DO
	MM := CONCAT(STR1:= '0', STR2:= MM);
END_WHILE;
WHILE LEN(DD) < 2 DO
	DD := CONCAT(STR1:= '0', STR2:= DD);
END_WHILE;
WHILE LEN(hh) < 2 DO
	hh := CONCAT(STR1:= '0', STR2:= hh);
END_WHILE;
WHILE LEN(Lmm) < 2 DO
	Lmm := CONCAT(STR1:= '0', STR2:= Lmm);
END_WHILE;
WHILE LEN(ss) < 2 DO
	ss := CONCAT(STR1:= '0', STR2:= ss);
END_WHILE;
WHILE LEN(xxx) < 3 DO
	xxx := CONCAT(STR1:= '0', STR2:= xxx);
END_WHILE;

TEMPSTRING := TimeFormat;

IF POS_YYYY <> 0 THEN
	TEMPSTRING := REPLACE(STR1:= TEMPSTRING, STR2:= YYYY, L:= 4, P:= POS_YYYY);
END_IF
IF POS_MM <> 0 THEN
	TEMPSTRING := REPLACE(STR1:= TEMPSTRING, STR2:= MM, L:= 2, P:= POS_MM);
END_IF
IF POS_DD <> 0 THEN
	TEMPSTRING := REPLACE(STR1:= TEMPSTRING, STR2:= DD, L:= 2, P:= POS_DD);
END_IF
IF POS_hh <> 0 THEN
	TEMPSTRING := REPLACE(STR1:= TEMPSTRING, STR2:= hh, L:= 2, P:= POS_hh);
END_IF
IF POS_Lmm <> 0 THEN
	TEMPSTRING := REPLACE(STR1:= TEMPSTRING, STR2:= Lmm, L:= 2, P:= POS_Lmm);
END_IF
IF POS_ss <> 0 THEN
	TEMPSTRING := REPLACE(STR1:= TEMPSTRING, STR2:= ss, L:= 2, P:= POS_ss);
END_IF
IF POS_xxx <> 0 THEN
	TEMPSTRING := REPLACE(STR1:= TEMPSTRING, STR2:= xxx, L:= 3, P:= POS_xxx);
END_IF
F_FormatTime := TEMPSTRING;

END_FUNCTION

// ---- TF11PlcSystem/System/Time/[obsolete]/Base_SysTime.TcPOU
(* 这个程序是一开始的时间获取程序，提供了两种时间源，将时间转换逻辑做在了内部。之后新写了一个功能块Base_SysInfo，将时间转换逻辑分开 *)
FUNCTION_BLOCK Base_SysTime
VAR_INPUT
	TimeSource : INT:=0; (* 0:systemInfo 1:FB_LocalSystemTime *)
END_VAR
VAR_OUTPUT
	oUnixTimeStamp10 : ULINT; (* 10位unix时间戳，代表从格林威治时间1970-01-01 00:00:00开始的秒数 *)
	oUnixTimeStamp13 : ULINT; (* 13位unix时间戳，代表从格林威治时间1970-01-01 00:00:00开始的秒数+3位毫秒数 *)
	oFileTime64 : T_FILETIME64; (* Utilities库中引入的Windows文件系统时间戳，代表从格林威治时间1601-01-01 00:00:00开始的纳秒数 *)
	oDateAndTime : DATE_AND_TIME; (* TwinCAT系统自带的本地时间日期格式，数值为10位unix时间戳，受到时区影响 *)
	oSystemTime : TIMESTRUCT; (* Utilities库中定义的本地时间日期格式，包含了年月日时分秒毫秒的结构体，受到时区影响 *)
	oTimeString : STRING;
	
END_VAR
VAR
	TimeZone : ULINT := 8;
	//TimeSource1
	SystemInfo : PlcAppSystemInfo;
	TaskInfo : PlcTaskSystemInfo;
	UnixTimeStamp10 : ULINT;
	UnixTimeStamp13 : ULINT;
	inFileTime64 : T_FILETIME64;
	
	
	//TimeSource2
	fbLocalSystemTime : FB_LocalSystemTime:=(sNetID:='', bEnable:=TRUE);
	localSystemTime :TIMESTRUCT;
	_fileTime64:T_FILETIME64;

END_VAR

CASE TimeSource OF
	0:(* TimeSource1 *)
	SystemInfo := _AppInfo;
	TaskInfo := _TaskInfo[GETCURTASKINDEXEX()];
	(* 946684800:从1970-2000年的秒数  11644473600:从1601-1970的秒数  5:误差补偿 *)
	(* DcTaskTime从2000-01-01 00:00:00:000开始，精确到1ns，10位Unix时间戳从1970-01-01 00:00:00开始，精确到1s *)
	UnixTimeStamp10 := 946684800 + LINT_TO_ULINT(TaskInfo.DcTaskTime)/1000000000;
	(* DcTaskTime从2000-01-01 00:00:00:000开始，精确到1ns，13位Unix时间戳从1970-01-01 00:00:00开始，精确到1ms *)
	UnixTimeStamp13 := 946684800_000 + LINT_TO_ULINT(TaskInfo.DcTaskTime)/1000000;
	(* FileTime64从1601-01-01 00:00:00开始，精确到100ns, *)
	inFileTime64 := LINT_TO_ULINT(TaskInfo.DcTaskTime)/100 + 946684800_0000000 + 11644473600_0000000 - 5_0000000;
	(* Output *)
	oUnixTimeStamp10 := UnixTimeStamp10;
	oUnixTimeStamp13 := UnixTimeStamp13;
	(* 将时间戳转换为自带的DATE_AND_TIME，要注意转换过来的是格林威治时间，需要加上8小时转换为北京时间 *)
	oDateAndTime:= ULINT_TO_DT(UnixTimeStamp10 + TimeZone * 3600 - 5);
	oFileTime64 := inFileTime64;
	(* 将时间戳转换为SYSTEM，要注意转换过来的是格林威治时间，需要加上8小时转换为北京时间 *)
	oSystemTime := FILETIME64_TO_SYSTEMTIME(inFileTime64 + TimeZone * 3600_0000000);

	1:
	//TimeSource2
	fbLocalSystemTime(bValid=> , systemTime=> localSystemTime, tzID=> );
	_fileTime64 := SYSTEMTIME_TO_FILETIME64(localSystemTime) - TimeZone * 36000000000;
	(* Output *)
	oSystemTime := localSystemTime;
	(* 因为Source2的时间源受到时区影响，所以都要减去时区 *)
	oFileTime64 := _fileTime64 ;
	oUnixTimeStamp13 := _fileTime64/10000 - 11644473600000  + 5000;
	oUnixTimeStamp10 := _fileTime64/10000000 - 11644473600  + 5;
	oDateAndTime := FILETIME64_TO_DT(_fileTime64 + TimeZone * 3600_0000000);
	
END_CASE

END_FUNCTION_BLOCK

// ---- TF11PlcSystem/System/Time/[obsolete]/FB_TimeConvertor0.TcPOU
{attribute 'hide_all_locals'}
(* 用于在多种常用的时间格式间进行转换的功能块,不考虑时区 *)
FUNCTION_BLOCK FB_TimeConvertor0
VAR_INPUT
	InputType : UDINT := 0 ; (* 0:DcTaskTime 1:10位Unix 2:13位Unix 3:FileTime64 4:DateAndTime 5:SystemTime *)
	iDcTaskTime : LINT; (* DcTaskTime从2000-01-01 00:00:00:000开始，精确到1ns *)
	iUnixTimeStamp10 : ULINT; (* 10位unix时间戳，代表从格林威治时间1970-01-01 00:00:00开始的秒数 *)
	iUnixTimeStamp13 : ULINT; (* 13位unix时间戳，代表从格林威治时间1970-01-01 00:00:00开始的秒数+3位毫秒数 *)
	iFileTime64 : T_FILETIME64; (* Utilities库中引入的Windows文件系统时间戳，代表从格林威治时间1601-01-01 00:00:00开始的纳秒数 *)
	iDateAndTime : DATE_AND_TIME; (* TwinCAT系统自带的本地时间日期格式，数值为10位unix时间戳，受到时区影响 *)
	iSystemTime : TIMESTRUCT; (* Utilities库中定义的本地时间日期格式，包含了年月日时分秒毫秒的结构体，受到时区影响 *)
END_VAR
VAR_OUTPUT
	oDcTaskTime : LINT;(* DcTaskTime从2000-01-01 00:00:00:000开始，精确到1ns *)
	oUnixTimeStamp10 : ULINT; (* 10位unix时间戳，代表从格林威治时间1970-01-01 00:00:00开始的秒数 *)
	oUnixTimeStamp13 : ULINT; (* 13位unix时间戳，代表从格林威治时间1970-01-01 00:00:00开始的秒数+3位毫秒数 *)
	oFileTime64 : T_FILETIME64; (* Utilities库中引入的Windows文件系统时间戳，代表从格林威治时间1601-01-01 00:00:00开始的纳秒数 *)
	oDateAndTime : DATE_AND_TIME; (* TwinCAT系统自带的本地时间日期格式，数值为10位unix时间戳，受到时区影响 *)
	oSystemTime : TIMESTRUCT; (* Utilities库中定义的本地时间日期格式，包含了年月日时分秒毫秒的结构体，受到时区影响 *)
	oStringTime : STRING(23); (* 时间字符串，年月日时分秒毫秒 *)
	oStringDate : STRING(10); (* 时间字符串，年月日 *)
	oStringTimeOfDay : STRING(12); (* 时间字符串，时分秒毫秒 *)
END_VAR
VAR
	(* 0 *)
	_in0DcTaskTime : LINT;(* DcTaskTime从2000-01-01 00:00:00:000开始，精确到1ns *)
	_in0UnixTimeStamp10 : ULINT; (* 10位unix时间戳，代表从格林威治时间1970-01-01 00:00:00开始的秒数 *)
	_in0UnixTimeStamp13 : ULINT; (* 13位unix时间戳，代表从格林威治时间1970-01-01 00:00:00开始的秒数+3位毫秒数 *)
	_in0FileTime64 : T_FILETIME64; (* Utilities库中引入的Windows文件系统时间戳，代表从格林威治时间1601-01-01 00:00:00开始的纳秒数 *)
	_in0DateAndTime : DATE_AND_TIME; (* TwinCAT系统自带的本地时间日期格式，数值为10位unix时间戳，受到时区影响 *)
	_in0SystemTime : TIMESTRUCT; (* Utilities库中定义的本地时间日期格式，包含了年月日时分秒毫秒的结构体，受到时区影响 *)
	(* string *)
	_in0StringTime : STRING(23); (* Utilities库中定义的本地时间日期格式，包含了年月日时分秒毫秒的结构体，受到时区影响 *)
	
	
END_VAR

(* 测试数据751214127491000000,1697898927,1697898927491,LDT#2023-10-21-14:35:22.491,DT#2023-10-21-14:35:22,..  *)
(* 由于Utilities库中自带了Filetime64与DT, Systemtime之间的转换，本功能块仅仅是添加了Filetime64与DcTaskTime与UnixTimeStamp之前的转换 *)
(* 转换思路是先尽可能转换成Filetime64，再利用自带函数转换 *)
(* Filetime64与DcTaskTime与UnixTimeStamp都是一种时间戳，区别在于起始时间或精度各不相同 *)
(* DcTaskTime从2000-01-01 00:00:00:000开始，精确到1ns *)
(* 10位Unix时间戳从1970-01-01 00:00:00开始，精确到1s，13位Unix时间戳加了三位表示毫秒的数 *)
(* FileTime64从1601-01-01 00:00:00开始，精确到100ns, *)
(* 946684800:从1970-2000年的秒数  11644473600:从1601-1970的秒数  5:误差补偿 *)
CASE InputType OF
	0:(* DcTaskTime从2000-01-01 00:00:00:000开始，精确到1ns *)
	(* Input *)
	_in0DcTaskTime := iDcTaskTime;
	(* Convert *)
	_in0FileTime64 := LINT_TO_ULINT(_in0DcTaskTime)/100 + 946684800_0000000 + 11644473600_0000000 - 5_0000000;
	_in0UnixTimeStamp13 := _in0FileTime64/10000 + 5000 - 11644473600000;
	_in0UnixTimeStamp10 := _in0UnixTimeStamp13 / 1000;
	_in0DateAndTime := FILETIME64_TO_DT(_in0FileTime64);
	_in0SystemTime := FILETIME64_TO_SYSTEMTIME(_in0FileTime64);
	
	1: (* Unix10 -> Unix13 : 由于10位时间戳不包含毫秒，所以转换出来的也不包含 *)
	(* Input *)
	_in0UnixTimeStamp10 := iUnixTimeStamp10;
	(* Convert *)
	_in0UnixTimeStamp13 := _in0UnixTimeStamp10 * 1000;
	_in0FileTime64 := (_in0UnixTimeStamp13 + 11644473600000 - 5000) * 10000;
	_in0DateAndTime := FILETIME64_TO_DT(_in0FileTime64);
	_in0SystemTime := FILETIME64_TO_SYSTEMTIME(_in0FileTime64);
	_in0DcTaskTime := ULINT_TO_LINT(_in0FileTime64 - 946684800_0000000 - 11644473600_0000000 + 5_0000000) * 100;
	
	2:
	(* Input *)
	_in0UnixTimeStamp13 := iUnixTimeStamp13;
	(* Convert *)
	_in0UnixTimeStamp10 := _in0UnixTimeStamp13 / 1000;
	_in0FileTime64 := (_in0UnixTimeStamp13 + 11644473600000 - 5000) * 10000;
	_in0DateAndTime := FILETIME64_TO_DT(_in0FileTime64);
	_in0SystemTime := FILETIME64_TO_SYSTEMTIME(_in0FileTime64);
	_in0DcTaskTime := ULINT_TO_LINT(_in0FileTime64 - 946684800_0000000 - 11644473600_0000000 + 5_0000000) * 100;
	
	3:
	(* Input *)
	_in0FileTime64 := iFileTime64;
	(* Convert *)
	_in0UnixTimeStamp13 := _in0FileTime64/10000 + 5000 - 11644473600000;
	_in0UnixTimeStamp10 := _in0UnixTimeStamp13 / 1000;
	_in0DateAndTime := FILETIME64_TO_DT(_in0FileTime64);
	_in0SystemTime := FILETIME64_TO_SYSTEMTIME(_in0FileTime64);
	_in0DcTaskTime := ULINT_TO_LINT(_in0FileTime64 - 946684800_0000000 - 11644473600_0000000 + 5_0000000) * 100;
	
	4:
	(* Input *)
	_in0DateAndTime := iDateAndTime;
	(* Convert *)
	_in0FileTime64 := DT_TO_FILETIME64(_in0DateAndTime);
	_in0UnixTimeStamp13 := _in0FileTime64/10000 + 5000 - 11644473600000;
	_in0UnixTimeStamp10 := _in0UnixTimeStamp13 / 1000;
	_in0SystemTime := FILETIME64_TO_SYSTEMTIME(_in0FileTime64);
	_in0DcTaskTime := ULINT_TO_LINT(_in0FileTime64 - 946684800_0000000 - 11644473600_0000000 + 5_0000000) * 100;
	
	5:
	(* Input *)
	_in0SystemTime :=iSystemTime;
	(* Convert *)
	_in0FileTime64 := SYSTEMTIME_TO_FILETIME64(_in0SystemTime);
	_in0UnixTimeStamp13 := _in0FileTime64/10000 + 5000 - 11644473600000;
	_in0UnixTimeStamp10 := _in0UnixTimeStamp13 / 1000;
	_in0DateAndTime := FILETIME64_TO_DT(_in0FileTime64);
	_in0DcTaskTime := ULINT_TO_LINT(_in0FileTime64 - 946684800_0000000 - 11644473600_0000000 + 5_0000000) * 100;
	
END_CASE
(* 2023-10-21 15:18:31:771 *)
_in0StringTime := F_SYSTEMTIME_TO_String6(_in0SystemTime, '');
oStringDate := MID(STR:= _in0StringTime, LEN:= 10, POS:= 1);
oStringTimeOfDay := MID(STR:= _in0StringTime, LEN:= 12, POS:= 12);
(* Output *)
oDcTaskTime := _in0DcTaskTime;
oUnixTimeStamp10 := _in0UnixTimeStamp10;
oUnixTimeStamp13 := _in0UnixTimeStamp13;
oFileTime64 := _in0FileTime64;
oDateAndTime := _in0DateAndTime;
oSystemTime := _in0SystemTime;
oStringTime := _in0StringTime;

END_FUNCTION_BLOCK

// ---- TF11PlcSystem/System/Time/[obsolete]/F_TimeStamp13_TO_SYSTEMTIME.TcPOU
FUNCTION F_TimeStamp13_TO_SYSTEMTIME : TimeStruct
VAR_INPUT
	iUnixTimeStamp13 : ULINT;
END_VAR
VAR
	_FileTime64 :T_FILETIME64;
END_VAR

_FileTime64 := (iUnixTimeStamp13 + 11644473600000 - 5000) * 10000;
F_TimeStamp13_TO_SYSTEMTIME := FILETIME64_TO_SYSTEMTIME(_FileTime64);

END_FUNCTION

// ---- TF11PlcSystem/System/Time/[obsolete]/PulseWrong.TcPOU
{attribute 'no_check'}
(* 脉冲生成器 Pulse Generator *)
FUNCTION_BLOCK PulseWrong
VAR_INPUT
	Enable : BOOL; (* BOOL, 启用脉冲生成器 *)
	Time_On : TIME; (* TIME, On脉冲时间 *)
	Time_Off : TIME; (* TIME, Off脉冲时间 *)
END_VAR
VAR_OUTPUT
	Q : BOOL; (* BOOL, 脉冲输出 *)
	RT : BOOL; (* BOOL, 脉冲输出上升沿 *)
	FT : BOOL; (* BOOL, 脉冲输出下降沿 *)
END_VAR
VAR
	tonPluse :TON;
END_VAR

(* 
Title		: 脉冲生成器 Pulse Generator
Time		: 2023-11-03
Creator		: Ulysses
Reference	: IOTA_Program
Commecnts	: 这个程序生成的脉冲会受到扫描周期的影响，每次脉冲都会偏移两个扫描周期
*)
(* 复位输出 *)
RT := FT := FALSE;
(* 内部逻辑 *)
IF Q AND (tonPluse.Q OR NOT Enable) THEN
	tonPluse(IN:= FALSE, PT:= Time_Off, Q=> , ET=> );
	FT := Q;
	Q := FALSE;
ELSIF NOT Q AND tonPluse.Q OR_ELSE Enable AND NOT tonPluse.IN THEN
	RT := NOT Q;
	tonPluse(IN:= FALSE, PT:= Time_On, Q=> , ET=> );
	Q := TRUE;
END_IF

tonPluse(IN:= Enable, PT:= , Q=> , ET=> );

END_FUNCTION_BLOCK
